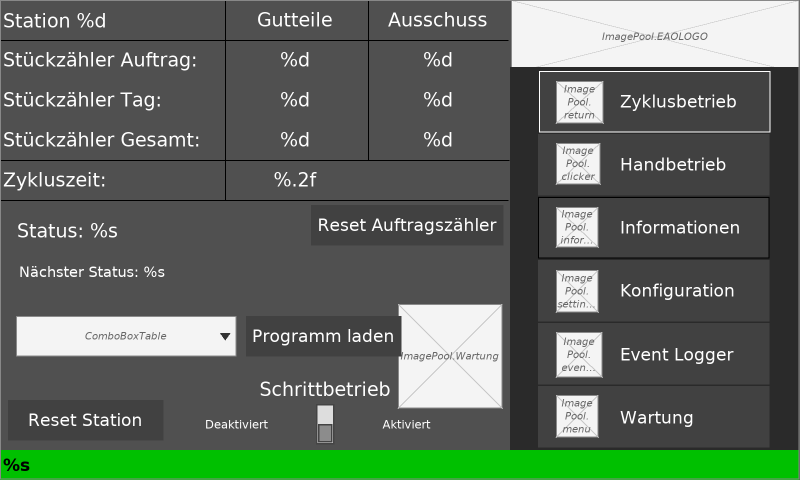
VISUALIZATION Zyklusbetrieb  // 800x480
    Textfield (0,40 225x40), "Stückzähler Auftrag:"
    Image (511,0 288x73), image: ImagePool.EAOLOGO
    Rectangle (510,67 289x412)
    Line (1,160) (509,160)
    Line (225,0) (225,200)
    Line (0,40) (508,40)
    Textfield (0,80 225x40), "Stückzähler Tag:"
    Textfield (0,120 225x40), "Stückzähler Gesamt:"
    Textfield (225,40 140x40), "%d", text variable: MAIN.stStueckzaehler.nGutteileAuftrag
    Line (368,0) (368,160)
    Textfield (225,80 140x40), "%d", text variable: MAIN.stStueckzaehler.nGutteileTag
    Textfield (225,120 140x40), "%d", text variable: MAIN.stStueckzaehler.nGutteileGesamt
    Textfield (368,80 140x40), "%d", text variable: MAIN.stStueckzaehler.nAusschussTag
    Textfield (368,40 140x40), "%d", text variable: MAIN.stStueckzaehler.nAusschussAuftrag
    Textfield (368,120 140x40), "%d", text variable: MAIN.stStueckzaehler.nAusschussGesamt
    Textfield (225,0 140x40), "Gutteile"
    Textfield (368,0 140x40), "Ausschuss"
    Rectangle (0,450 799x30), "%s", text variable: MAIN.HMI.sStatus, colour variable: MAIN.HMI.nColorInfoBalken
        p3450524324: MAIN.HMI.nColorInfoBalken
    Line (0,200) (508,200)
    Textfield (0,160 225x40), "Zykluszeit:"
    Textfield (225,160 140x40), "%.2f", text variable: MAIN.fbZyklusZeitGesamt.fZyklusZeit
    RoundedRectangle (8,400 155x40), "Reset Station"
        OnMouseClick: execute { MAIN.fbSt1.bBtnReset := TRUE; }
    Textfield (0,1 140x40), "Station %d", text variable: MAIN.HMI.nAnzeigeStation
    Textfield (14,211 225x40), "Status: %s", text variable: MAIN.HMI.sStationStatus
    Rectangle (539,71 231x61)
        OnMouseClick: change screen: Zyklusbetrieb
    Textfield (617,71 153x61), "Zyklusbetrieb"
        OnMouseClick: change screen: Zyklusbetrieb
    Rectangle (538,134 231x61)
        OnMouseClick: change screen: Handbetrieb
    Textfield (617,134 153x61), "Handbetrieb"
        OnMouseClick: change screen: Handbetrieb
    Image (556,143 44x41), image: ImagePool.clicker
        OnMouseClick: change screen: Handbetrieb
    Image (556,81 47x42), image: ImagePool.return
        OnMouseClick: change screen: Zyklusbetrieb
    Rectangle (538,197 231x61)
        OnMouseClick: change screen: Diagnose
    Textfield (617,197 153x61), "Informationen"
        OnMouseClick: change screen: Diagnose
    Image (556,207 42x40), image: ImagePool.information
        OnMouseClick: change screen: Diagnose
    Rectangle (538,323 231x61)
        OnMouseClick: change screen: EventLogger
    Textfield (617,324 153x61), "Event Logger"
        OnMouseClick: change screen: EventLogger
    Image (556,332 46x45), image: ImagePool.eventLogger
        OnMouseClick: change screen: EventLogger
    Rectangle (538,260 231x61)
        OnMouseClick: change screen: Konfig1
    Textfield (617,260 153x61), "Konfiguration"
        OnMouseClick: change screen: Konfig1
    Image (556,270 42x42), image: ImagePool.settings
        OnMouseDown: change screen: Konfig1
    Rectangle (538,386 231x61)
        OnMouseClick: change screen: Wartung
    Textfield (617,387 153x61), "Wartung"
        OnMouseClick: change screen: Wartung
    Image (556,395 42x42), image: ImagePool.menu
        OnMouseDown: change screen: Wartung
    Image (398,304 104x104), invisible if: NOT MAIN.fbSt1.bWarnungNothalt, image: ImagePool.Wartung
        OnMouseDown: change screen: Wartung
    RoundedRectangle (311,205 192x40), "Reset Auftragszähler"
        OnMouseClick: execute { MAIN.fbSt1.bBtnResetAuftrZaehler := TRUE; }
    ComboBoxTable (16,316 220x40), variable: MAIN.HMI.nAngewaehltesProg, data array: MAIN.HMI.aProgrammNamen
        p3854506369: MAIN.HMI.aProgrammNamen[INDEX]
        p1892666644: MAIN.HMI.aProgramm[INDEX].sName
        p338671338: MAIN.HMI.aProgramm[INDEX].aAktorBew
        p1128707560: Parameter.cMaxProgramme
    RoundedRectangle (246,316 155x40), "Programm laden", colour toggle: MAIN.HMI.bProgrammGeladen, input disabled if: MAIN.HMI.bProgeammLadenBtnInaktiv
        OnMouseClick: execute { MAIN.HMI.bBtnProgrammLaden := TRUE; }
    Textfield (200,399 73x51), "Deaktiviert"
    Textfield (225,375 200x29), "Schrittbetrieb"
    Textfield (370,399 73x51), "Aktiviert"
    DipSwitch (280,404 90x40), variable: MAIN.HMI.bBtnSchrittbetrieb, behaviour: TOGGLE, style: Switch-DipSwitch-Gray
    Textfield (16,252 225x40), "Nächster Status: %s", text variable: MAIN.fbSt1.sNaechsterSchritt, invisible if: not MAIN.fbSt1.bSchrittbetriebAktiv
END_VISUALIZATION

(* stored: Version 1.1.0.1, ProductVersion 3.1.4024.12
   Visu Zyklusbetrieb: Id {ffc19b42-ac78-478b-b509-10af9a59899c} *)
